{attribute 'linkalways'}
{attribute 'hide_all_locals'}
FUNCTION_BLOCK ValueLint EXTENDS ValueLintRead IMPLEMENTS Value
VAR
END_VAR

METHOD SetFromType : BOOL
VAR_INPUT
	source : __SYSTEM.AnyType;
END_VAR
SetFromType := ConvertAnyType(source, thisAnyType);
END_METHOD

METHOD SetFromString : BOOL
VAR_INPUT
	value : T_MaxString;
END_VAR
thisValue := STRING_TO_LINT(value);

SetFromString := TRUE;
END_METHOD

METHOD Set : BOOL
VAR_INPUT
	source : ANY;
END_VAR
Set := ConvertAnyType(source, thisAnyType);
END_METHOD

END_FUNCTION_BLOCK

(* stored: Version 1.1.0.1
   POU ValueLint: Id {8d2574c7-bb99-45f5-b503-fe2cd66cb02f}, SpecialFunc None
   Method SetFromType: Id {91837268-9abe-4370-adee-0062503aed48}
   Method SetFromString: Id {9b61d5bf-177b-4f09-b1bf-a3ab41c976f0}
   Method Set: Id {cae9570f-1c18-41e2-a141-f95c2da65918} *)
